// TIA Portal V19 export
TYPE "UDT_VALVEFAULTS"
   STRUCT
      ctrl : Struct   // External data (Primary alarm data - alarm & plc ackn)
         alarm_ftamain : Bool := false;
         alarm_ftaupper : Bool := false;
         alarm_ftalower : Bool := false;
         alarm_ftd : Bool := false;
         bit12 : Bool := false;
         alarm_il : Bool := false;
         bit14 : Bool := false;
         bit15 : Bool := false;
         plcackn_ftamain : Bool := false;
         plcackn_ftaupper : Bool := false;
         plcackn_ftalower : Bool := false;
         plcackn_ftd : Bool := false;
         bit4 : Bool := false;
         plcackn_il : Bool := false;
         bit6 : Bool := false;
         bit7 : Bool := false;
      END_STRUCT;
      status : Struct   // External data (Secondary alarm data - siren & hmi ackn)
         siren_ftamain : Bool := false;
         siren_ftaupper : Bool := false;
         siren_ftalower : Bool := false;
         siren_ftd : Bool := false;
         bit12 : Bool := false;
         siren_il : Bool := false;
         bit14 : Bool := false;
         bit15 : Bool := false;
         hmiackn_ftamain : Bool := false;
         hmiackn_ftaupper : Bool := false;
         hmiackn_ftalower : Bool := false;
         hmiackn_ftd : Bool := false;
         bit4 : Bool := false;
         hmiackn_il : Bool := false;
         bit6 : Bool := false;
         bit7 : Bool := false;
      END_STRUCT;
   END_STRUCT;
END_TYPE
